(* CODESYS project Simple Socket Communication.project

Project tree, tasks and I/O mapping:
  Device : CODESYS Control for Raspberry Pi, 3S - Smart Software Solutions GmbH, version 3.5.11.20
    application Application
      libraries: Standard, * (System); Network, 3.5.7.0 (3S - Smart Software Solutions GmbH); Raspberry I2C Gyroscopes, 1.1.1.0 (3S - Smart Software Solutions GmbH)
      task MainTask (cyclic, interval 4 ms, priority 1) calls PLC_PRG
      task VISU_TASK (cyclic, interval 100 ms, priority 31) calls VisuElems.Visu_Prg
      program PLC_PRG [CFC]
      function block SocketVerbindung [ST]
      visualisation Visualization
    SoftMotion General Axis Pool
    I²C
    SPI
    GPIOs_A_B : GPIOs A/B, 3S - Smart Software Solutions GmbH, version 3.5.11.0
        unmapped channels: digital inputs (GPIO0..GPIO31), digital outputs (GPIO0..GPIO31)
    Onewire
    Camera device
      <Leer>
  text list GlobalTextList
*)

// Device/Application/PLC_PRG
PROGRAM PLC_PRG
VAR
	NeuerSocket: SocketVerbindung;
	taster: BOOL;
	ip: STRING := '192.168.24.3';
END_VAR

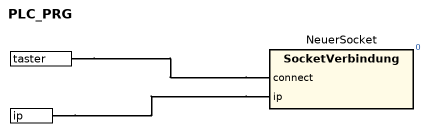
NeuerSocket(connect := taster, ip := ip); // SocketVerbindung

END_PROGRAM

// Device/Application/SocketVerbindung
FUNCTION_BLOCK SocketVerbindung
VAR_INPUT
	connect: BOOL;
	ip: STRING;
	port: UINT := 4444;
END_VAR
VAR_OUTPUT
END_VAR
VAR
 	address: NBS.SOCKADDRESS;
	inaddr : nbs.INADDR;
 	send: STRING := 'hello';
 	receive: STRING;
 	objectArray: ARRAY[0..6] OF REAL;
	pResult: POINTER TO NBS.RTS_IEC_RESULT;
	pResult2: NBS.RTS_IEC_RESULT; 
	pInAddr: POINTER TO UDINT;
 
 	result: UDINT;
 	socketId: nbs.RTS_IEC_HANDLE;
 	terminate: BOOL;
	sin_addr: UDINT;
	
	step_no: INT;
	timeout: TON;
	sendBytes: __XINT;
END_VAR


CASE step_no OF

	0: 
		IF connect THEN
			step_no := 10;
		END_IF;
		
	10: 
		pResult2 := nbs.SysSockInetAddr(ip, ADR(inaddr));
		address.sin_addr := inaddr;
		address.sin_family := NBS.SOCKET_AF_INET;
		address.sin_port := nbs.syssockhtons(port);
		
		IF socketId = 0 AND terminate = FALSE THEN (* Verbindung aufbauen *)
		  	socketId := NBS.SysSockCreate(NBS.SOCKET_AF_INET, NBS.SOCKET_STREAM, 0, pResult);
		  	result := NBS.SysSockConnect(socketId, ADR(address), SIZEOF(address));
		ELSE
		 	IF terminate = TRUE THEN (* Verbindung abbauen *)
		  		nbs.SysSockClose(socketId);
		  		socketId := 0;
		  		result := 0;
		 	END_IF (* Verbunden *) 
		END_IF
		
		sendBytes := nbs.SysSockSend(socketId, ADR(send), SIZEOF(send), 1, pResult); 
		 //nbs.SysSockRecv(socketId, ADR(receive), SIZEOF(receive), 1);
		 //objectArray := split(receive);
		
		step_no := 20;
		
	20:
		timeout(IN:=TRUE, PT:=T#5S);
		IF timeout.Q THEN
			timeout(IN:=FALSE, PT:=T#5S);
			step_no := 0;
		END_IF

END_CASE

END_FUNCTION_BLOCK

// Device/Application/Visualization
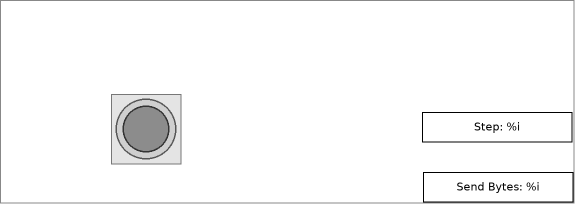
VISUALIZATION Visualization  // 575x204
    PushSwitch (111,94 70x70), variable: PLC_PRG.taster, behaviour: TAP, style: Switch-PushSwitch-Gray
    Rectangle (422,112 150x30), "Step: %i", text variable: PLC_PRG.NeuerSocket.step_no
    Rectangle (423,172 150x30), "Send Bytes: %i", text variable: PLC_PRG.NeuerSocket.sendBytes
END_VISUALIZATION
